# EPICS alarm handler configuration: apps/alhConfig/svt.alhConfig
#===============================================================================
# SVT Alarm Config
#===============================================================================

GROUP NULL SVT

INCLUDE SVT /usr/clas12/hps/prod/apps/alhConfig/svtVoltage.alhConfig
INCLUDE SVT /usr/clas12/hps/prod/apps/alhConfig/svtCooling.alhConfig
